Yaskawa INFORM job: half_bracket_cylinder_program.JBI

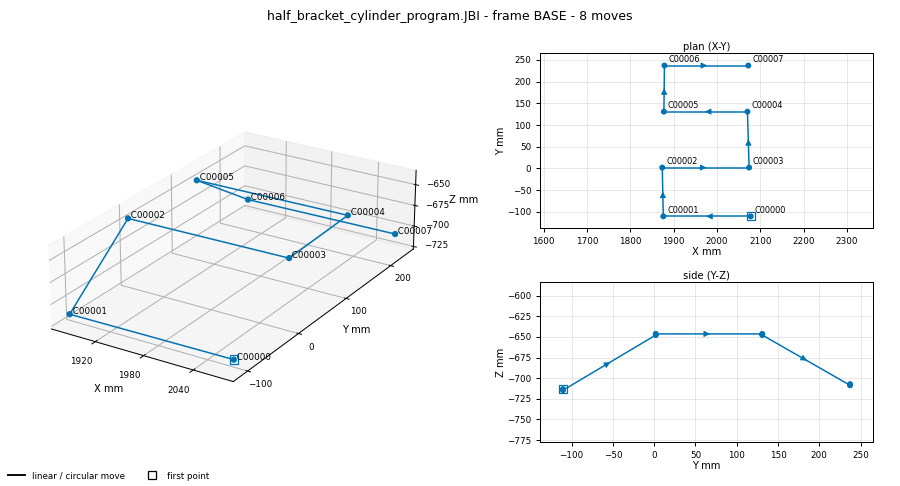
[picture p0: tool path of half_bracket_cylinder_program.JBI in frame BASE, 8 of 11 moves have a stored position in this frame; points joined in program order, loops and branches not executed]
/JOB
//NAME half_bracket_cylinder_program
//POS
///NPOS 8,0,8,0,0,0
///TOOL 0
///POSTYPE BASE
///RECTAN
///RCONF 0,0,0,0,0,0,0,0,0,0,0,0,0,0,0,0,0,0,0,0,0,0,0,0
C00000=2077.796056,-110.551507,-713.190901,175.000000,-46.257803,89.627835
C00001=1876.144105,-110.551512,-714.559538,175.000000,-46.257803,89.627835
C00002=1873.788855,1.921201,-647.646927,-164.746246,-5.000000,-5.000000
C00003=2074.054674,1.921206,-646.287698,-164.746246,-5.000000,-5.000000
C00004=2070.212979,130.856473,-646.342400,164.720803,-5.000000,5.000000
C00005=1877.558074,130.856468,-647.649973,164.720803,-5.000000,5.000000
C00006=1878.780911,237.253182,-708.515135,-175.000000,-44.272579,-89.601120
C00007=2072.217866,237.253186,-707.202254,-175.000000,-44.272579,-89.601120
///POSTYPE PULSE
///PULSE
EX00000=188416.0
///POSTYPE PULSE
///PULSE
EC00000=188416.0
EC00001=188416.0
EC00002=188416.0
EC00003=188416.0
EC00004=188416.0
EC00005=188416.0
EC00006=188416.0
EC00007=188416.0
//INST
///DATE 2023/08/15 15:25
///ATTR SC,RW,RJ
////FRAME BASE
///GROUP1 RB1,ST1
NOP
MOVJ P009 EX000 VJ=15.00
MOVJ C00000 EC00000 VJ=15.0
CALL JOB:SPYON
MOVL C00001 EC00001 V=150.0
MOVL C00002 EC00002 V=150.0
MOVL C00003 EC00003 V=150.0
MOVL C00004 EC00004 V=150.0
MOVL C00005 EC00005 V=150.0
MOVL C00006 EC00006 V=150.0
MOVL C00007 EC00007 V=150.0
CALL JOB:SPYOF
MOVJ P009 VJ=15.00
MOVL P009 EX00000 V=150.0
END
